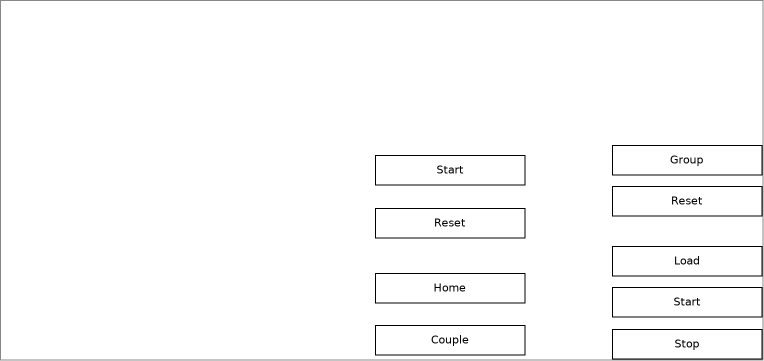
VISUALIZATION Visualization  // 764x361
    Rectangle (375,325 150x30), "Couple", colour toggle: MAIN.bGearIn
        toggle MAIN.bGearIn
    Rectangle (375,273 150x30), "Home"
        tap MAIN.bHome
    Rectangle (375,155 150x30), "Start", colour toggle: MAIN.bEN
        toggle MAIN.bEN
    Rectangle (375,208 150x30), "Reset", colour toggle: MAIN.bReset
        tap MAIN.bReset
    Rectangle (612,145 150x30), "Group", colour toggle: POU_NCI.bBuildGroup
        toggle POU_NCI.bBuildGroup
    Rectangle (612,186 150x30), "Reset"
        tap POU_NCI.bReset
    Rectangle (612,287 150x30), "Start"
        tap POU_NCI.bStart
    Rectangle (612,329 150x30), "Stop"
        tap POU_NCI.bStop
    Rectangle (612,246 150x30), "Load"
        tap POU_NCI.bLoad
END_VISUALIZATION

(* stored: Version 1.1.0.1, ProductVersion 3.1.4022.12
   Visu Visualization: Id {588864ef-d643-4503-9476-1744d0cbd0a7} *)
